% RSLogix 500 project HEATER PID CONTROL WITH ALARMS AND NOTIFICATIONS.RSS, saved by version 8.30.00.16 %
PROJECT "UNTITLED"    % processor: Bul.1763 MicroLogix 1100 Series B %

PROGRAM FILES
  LAD 2 "MAIN"  4 rungs
  LAD 3 "I/O"  5 rungs
  LAD 4 "CONTROLS"  2 rungs
  LAD 5 "ALARMS"  3 rungs

DATA FILES
  O0 OUTPUT  8 elements
  I1 INPUT  22 elements
  S2 STATUS  66 elements
  B3 BINARY  1 elements
  T4 TIMER  1 elements
  C5 COUNTER  1 elements
  R6 CONTROL  1 elements
  N7 INTEGER  2 elements
  F8 FLOAT  2 elements
  PD9 PID   1 elements

LADDER 2 "MAIN"
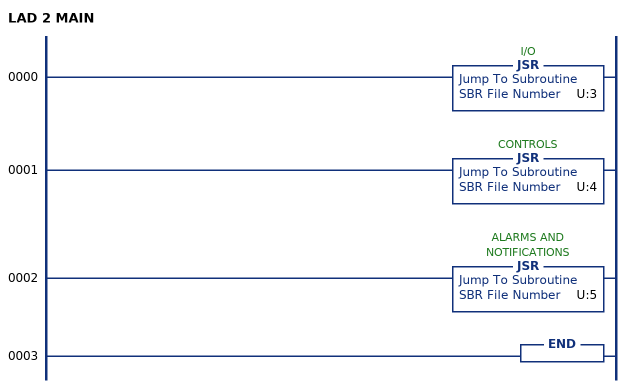
% Rung: 0 %
SOR JSR U:3 EOR
%   U:3  "I/O" %
% Rung: 1 %
SOR JSR U:4 EOR
%   U:4  "CONTROLS" %
% Rung: 2 %
SOR JSR U:5 EOR
%   U:5  "ALARMS AND NOTIFICATIONS" %
% Rung: 3 %
SOR END EOR

LADDER 3 "I/O"
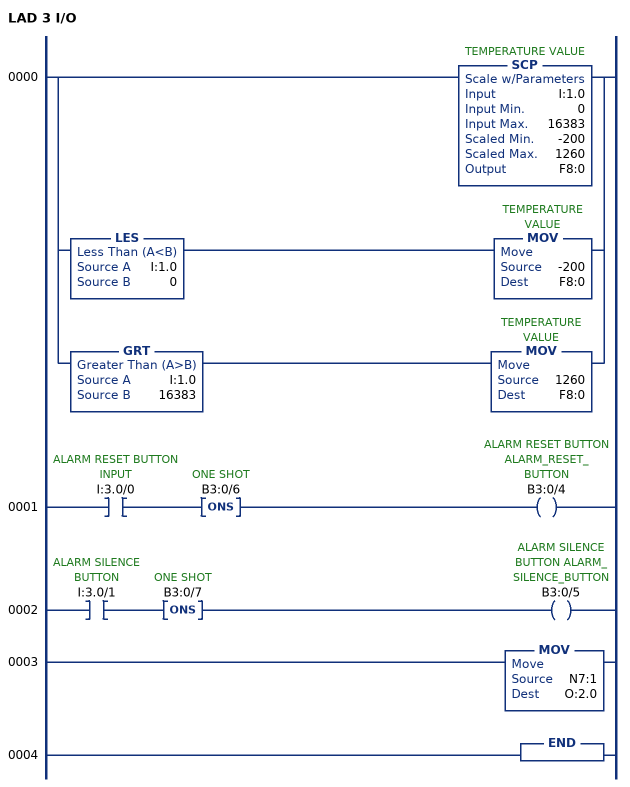
% Rung: 0 %
SOR BST SCP I:1.0 0 16383 -200 1260 F8:0 NXB LES I:1.0 0 MOV -200 F8:0 NXB GRT I:1.0 16383 MOV 1260 F8:0 BND EOR
%   F8:0  "TEMPERATURE VALUE" %
% Rung: 1 %
SOR XIC I:3.0/0 ONS B3:0/6 OTE B3:0/4 EOR
%   I:3.0/0  "ALARM RESET BUTTON INPUT" %
%   B3:0/6  "ONE SHOT" %
%   B3:0/4  ALARM_RESET_BUTTON  "ALARM RESET BUTTON" %
% Rung: 2 %
SOR XIC I:3.0/1 ONS B3:0/7 OTE B3:0/5 EOR
%   I:3.0/1  "ALARM SILENCE BUTTON" %
%   B3:0/7  "ONE SHOT" %
%   B3:0/5  ALARM_SILENCE_BUTTON  "ALARM SILENCE BUTTON" %
% Rung: 3 %
SOR MOV N7:1 O:2.0 EOR
% Rung: 4 %
SOR END EOR

LADDER 4 "CONTROLS"
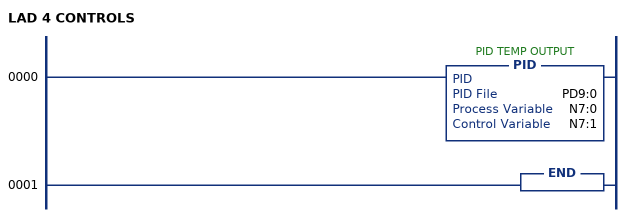
% Rung: 0 %
SOR PID PD9:0 N7:0 N7:1 EOR
%   PD9:0  "PID TEMP OUTPUT" %
%   N7:0  "TANK LEVEL" %
% Rung: 1 %
SOR END EOR

LADDER 5 "ALARMS"
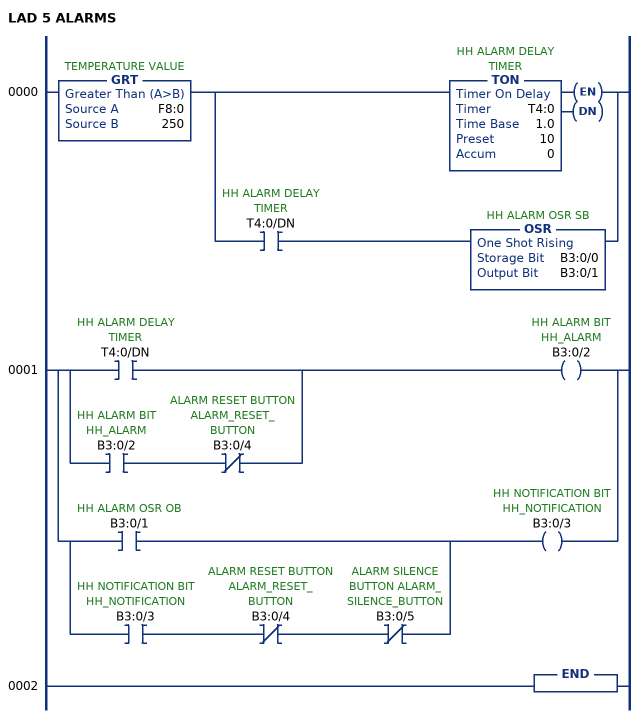
% Rung: 0 %
SOR GRT F8:0 250 BST TON T4:0 1.0 10 0 NXB XIC T4:0/DN OSR B3:0/0 B3:0/1 BND EOR
%   F8:0  "TEMPERATURE VALUE" %
%   T4:0  "HH ALARM DELAY TIMER" %
%   B3:0/0  "HH ALARM OSR SB" %
%   B3:0/1  "HH ALARM OSR OB" %
% Rung: 1 %
SOR BST BST XIC T4:0/DN NXB XIC B3:0/2 XIO B3:0/4 BND OTE B3:0/2 NXB BST XIC B3:0/1 NXB XIC B3:0/3 XIO B3:0/4 XIO B3:0/5 BND OTE B3:0/3 BND EOR
%   T4:0  "HH ALARM DELAY TIMER" %
%   B3:0/2  HH_ALARM  "HH ALARM BIT" %
%   B3:0/4  ALARM_RESET_BUTTON  "ALARM RESET BUTTON" %
%   B3:0/1  "HH ALARM OSR OB" %
%   B3:0/3  HH_NOTIFICATION  "HH NOTIFICATION BIT" %
%   B3:0/5  ALARM_SILENCE_BUTTON  "ALARM SILENCE BUTTON" %
% Rung: 2 %
SOR END EOR

OTHER DOCUMENTED ADDRESSES
  I:1.0/0  "K THERMOCOUPLE INPUT"
  T4:2/DN  "LL ALARM TIMER DN BIT"

DATA TABLE (non-zero values as saved)
DATA T4
% .PRE .ACC %
% T4:0 % 10 0
